% RSLogix 500 project REDA.RSS, saved by version 8.10.00.18 %
PROJECT "UNTITLED"    % processor: type code 157 %

PROGRAM FILES
  LAD 2   25 rungs

DATA FILES
  O0 OUTPUT  1 elements
  I1 INPUT  1 elements
  S2 STATUS  83 elements
  B3 BINARY  1 elements
  T4 TIMER  21 elements
  C5 COUNTER  1 elements
  R6 CONTROL  1 elements
  N7 INTEGER  1 elements
  F8 FLOAT  1 elements

LADDER 2
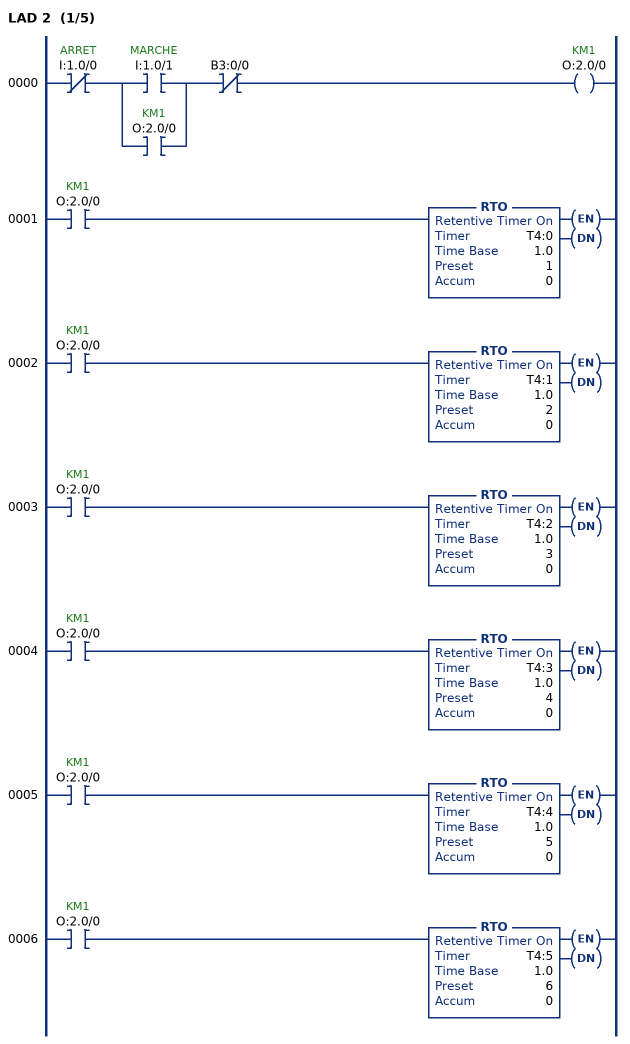
% Rung: 0 %
SOR XIO I:1.0/0 BST XIC I:1.0/1 NXB XIC O:2.0/0 BND XIO B3:0/0 OTE O:2.0/0 EOR
%   I:1.0/0  ARRET %
%   I:1.0/1  MARCHE %
%   O:2.0/0  KM1 %
% Rung: 1 %
SOR XIC O:2.0/0 RTO T4:0 1.0 1 0 EOR
%   O:2.0/0  KM1 %
% Rung: 2 %
SOR XIC O:2.0/0 RTO T4:1 1.0 2 0 EOR
%   O:2.0/0  KM1 %
% Rung: 3 %
SOR XIC O:2.0/0 RTO T4:2 1.0 3 0 EOR
%   O:2.0/0  KM1 %
% Rung: 4 %
SOR XIC O:2.0/0 RTO T4:3 1.0 4 0 EOR
%   O:2.0/0  KM1 %
% Rung: 5 %
SOR XIC O:2.0/0 RTO T4:4 1.0 5 0 EOR
%   O:2.0/0  KM1 %
% Rung: 6 %
SOR XIC O:2.0/0 RTO T4:5 1.0 6 0 EOR
%   O:2.0/0  KM1 %

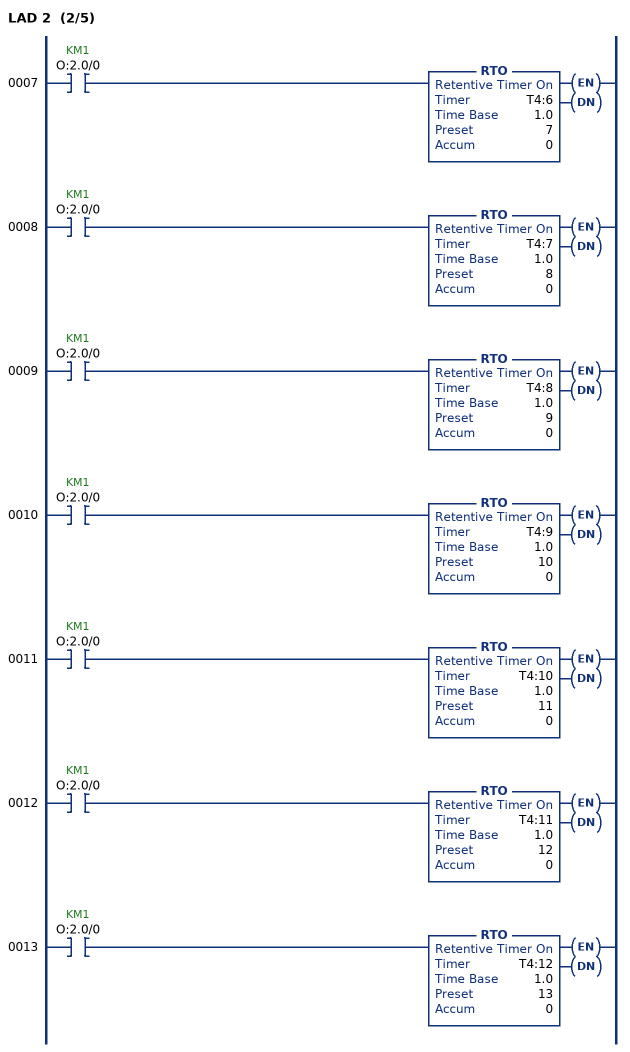
% Rung: 7 %
SOR XIC O:2.0/0 RTO T4:6 1.0 7 0 EOR
%   O:2.0/0  KM1 %
% Rung: 8 %
SOR XIC O:2.0/0 RTO T4:7 1.0 8 0 EOR
%   O:2.0/0  KM1 %
% Rung: 9 %
SOR XIC O:2.0/0 RTO T4:8 1.0 9 0 EOR
%   O:2.0/0  KM1 %
% Rung: 10 %
SOR XIC O:2.0/0 RTO T4:9 1.0 10 0 EOR
%   O:2.0/0  KM1 %
% Rung: 11 %
SOR XIC O:2.0/0 RTO T4:10 1.0 11 0 EOR
%   O:2.0/0  KM1 %
% Rung: 12 %
SOR XIC O:2.0/0 RTO T4:11 1.0 12 0 EOR
%   O:2.0/0  KM1 %
% Rung: 13 %
SOR XIC O:2.0/0 RTO T4:12 1.0 13 0 EOR
%   O:2.0/0  KM1 %

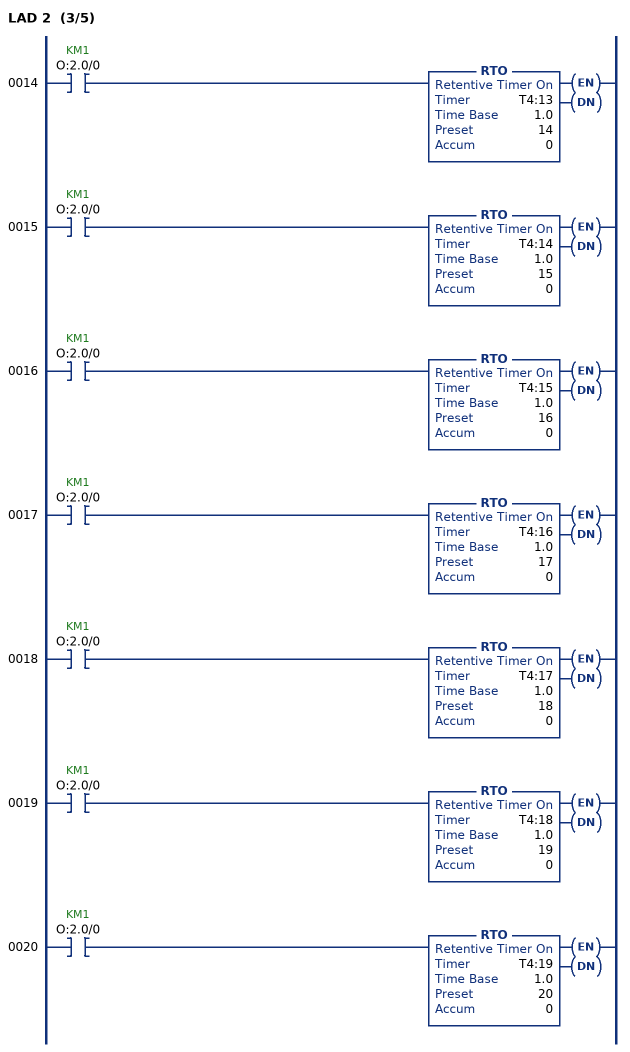
% Rung: 14 %
SOR XIC O:2.0/0 RTO T4:13 1.0 14 0 EOR
%   O:2.0/0  KM1 %
% Rung: 15 %
SOR XIC O:2.0/0 RTO T4:14 1.0 15 0 EOR
%   O:2.0/0  KM1 %
% Rung: 16 %
SOR XIC O:2.0/0 RTO T4:15 1.0 16 0 EOR
%   O:2.0/0  KM1 %
% Rung: 17 %
SOR XIC O:2.0/0 RTO T4:16 1.0 17 0 EOR
%   O:2.0/0  KM1 %
% Rung: 18 %
SOR XIC O:2.0/0 RTO T4:17 1.0 18 0 EOR
%   O:2.0/0  KM1 %
% Rung: 19 %
SOR XIC O:2.0/0 RTO T4:18 1.0 19 0 EOR
%   O:2.0/0  KM1 %
% Rung: 20 %
SOR XIC O:2.0/0 RTO T4:19 1.0 20 0 EOR
%   O:2.0/0  KM1 %

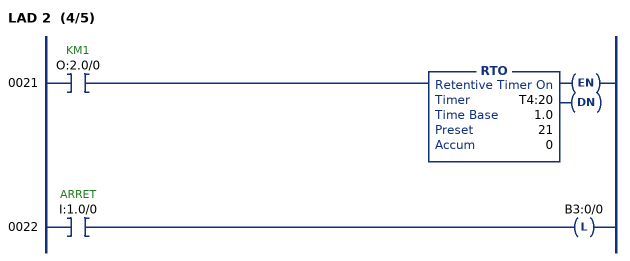
% Rung: 21 %
SOR XIC O:2.0/0 RTO T4:20 1.0 21 0 EOR
%   O:2.0/0  KM1 %
% Rung: 22 %
SOR XIC I:1.0/0 OTL B3:0/0 EOR
%   I:1.0/0  ARRET %

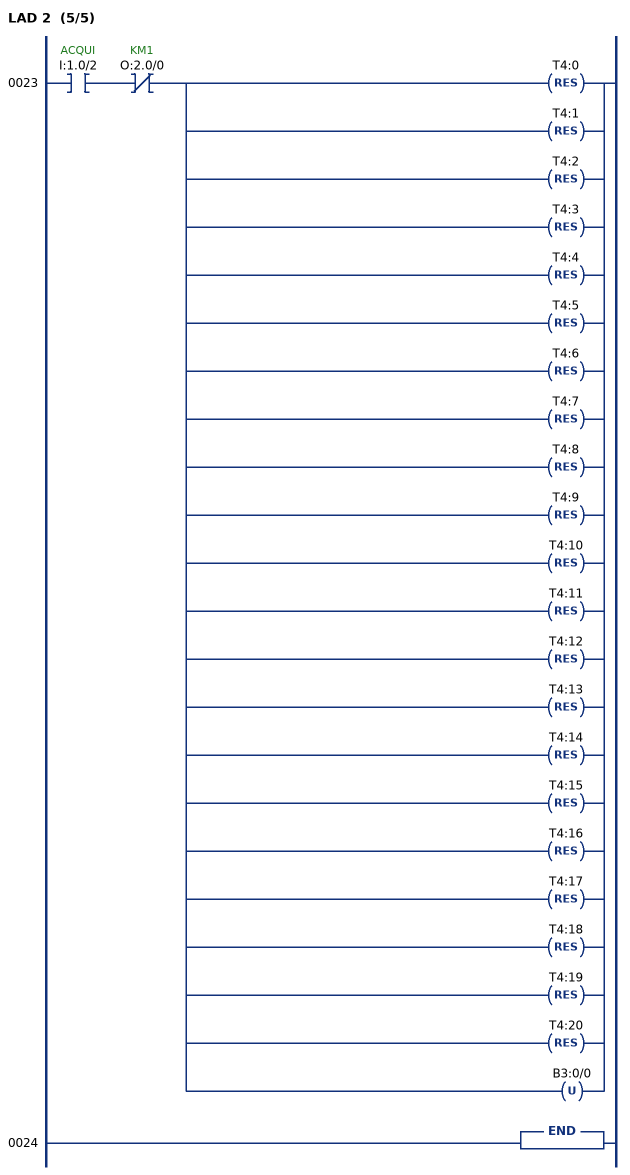
% Rung: 23 %
SOR XIC I:1.0/2 XIO O:2.0/0 BST RES T4:0 NXB RES T4:1 NXB RES T4:2 NXB RES T4:3 NXB RES T4:4 NXB RES T4:5 NXB RES T4:6 NXB RES T4:7 NXB RES T4:8 NXB RES T4:9 NXB RES T4:10 NXB RES T4:11 NXB RES T4:12 NXB BST RES T4:13 NXB RES T4:14 NXB RES T4:15 NXB RES T4:16 NXB RES T4:17 NXB RES T4:18 NXB RES T4:19 NXB RES T4:20 NXB OTU B3:0/0 BND BND EOR
%   I:1.0/2  ACQUI %
%   O:2.0/0  KM1 %
% Rung: 24 %
SOR END EOR

DATA TABLE (non-zero values as saved)
DATA T4
% .PRE .ACC %
% T4:0 % 1 0
% T4:1 % 2 0
% T4:2 % 3 0
% T4:3 % 4 0
% T4:4 % 5 0
% T4:5 % 6 0
% T4:6 % 7 0
% T4:7 % 8 0
% T4:8 % 9 0
% T4:9 % 10 0
% T4:10 % 11 0
% T4:11 % 12 0
% T4:12 % 13 0
% T4:13 % 14 0
% T4:14 % 15 0
% T4:15 % 16 0
% T4:16 % 17 0
% T4:17 % 18 0
% T4:18 % 19 0
% T4:19 % 20 0
% T4:20 % 21 0
